FUNCTION_BLOCK FB_NormallyClosedSensor IMPLEMENTS I_Sensor
VAR
	Input AT %I* : BOOL;
END_VAR

{warning 'add property implementation'}
PROPERTY IsActive : BOOL
GET
IsActive := NOT Input;
END_GET
END_PROPERTY

END_FUNCTION_BLOCK

(* stored: Version 1.1.0.1, ProductVersion 3.1.4024.9
   POU FB_NormallyClosedSensor: Id {767b69c1-a26c-49cb-9630-29aa8f94980c}, SpecialFunc None
   Property IsActive: Id {229e4f62-cff1-4d55-b269-5dd6ebb541b8}
   Get Get: Id {ac7cc2f5-984e-40b5-808b-b95b7da0fc30} *)
